// TIA Portal project "TCP Client" (V15.1)

(* hardware
DEVICE "ET 200SP station_1"  ET 200SP-Station
   slot 0: "Rack_0"  Rack  6ES5 710-8MAx1
   slot 1: "PLC_1"  CPU 1510SP F-1 PN  6ES7 510-1SJ00-0AB0  V1.8
   slot 127: "BA 2xRJ45"  BA 2xRJ45  6ES7 193-6AR00-0AA0  V0.0
      slot 32769: "Port_1"  6ES7 193-6AR00-0AA0
      slot 32770: "Port_2"  6ES7 193-6AR00-0AA0
*)

// ===== PLC "PLC_1"  CPU 1510SP F-1 PN =====

FUNCTION_BLOCK "01CommTCP"   // FB4, SCL
{ S7_Optimized_Access := 'FALSE' }
VERSION : 0.1
   VAR_INPUT
      IP1 : Byte;
      IP2 : Byte;
      IP3 : Byte;
      IP4 : Byte;
      Port : UInt;
      ConID : Conn_Ouc;
   END_VAR
   VAR
      RcvBusy : Bool;
      SndBuf : Array[1..40] of Char;
      RcvBuf : Array[1..40] of Char;
      Size : Struct
         Snd : Int;
         Rcv : Int;
      END_STRUCT;
      Connect : TCON;
      Snd : TSEND;
      Rcv : TRCV;
      SndCount : Int;
      RcvCount : Int;
      Req : Bool;
      RcvLen : Int;
      "Step" : Int;
      Zero : Int;
      RetVal : Int;
      Tout : TON_TIME;
      TON_Repeat : TON_TIME;
      DisConnect : TDISCON;
      conData : TCON_IP_v4;
      tonDelay : TON_TIME;
      tonConTout : TON_TIME;
      tonConWarning : TON_TIME;
      WarnConnection : Program_Alarm;
      wStatus : Word;
      byTestState : Byte;
      xError : Bool;
      CntOfSendBuf : UInt;
      CntOfRecBuf : UInt;
      bufferTimer : TON_TIME;
      status : Word;
      error : Bool;
   END_VAR
   VAR_TEMP
      xSig : Bool;
   END_VAR
BEGIN
   //********************************************************************************
   // Initialization
   //********************************************************************************

   CASE #Step OF

   0:
       //*********************************
       //  Init part 1 step moved to 0
       //*********************************
       #conData.InterfaceId := 64;
       #conData.ID := #ConID;
       #conData.ConnectionType := 11;
       #conData.ActiveEstablished := True;
       #conData.RemotePort := #Port;
       #conData.LocalPort := 0;
       #conData.RemoteAddress.ADDR[1] := #IP1;
       #conData.RemoteAddress.ADDR[2] := #IP2;
       #conData.RemoteAddress.ADDR[3] := #IP3;
       #conData.RemoteAddress.ADDR[4] := #IP4;
       #Step := 1;

   1:  //*********************************
       //  Init Part 2
       //*********************************
       #RcvCount := 0;
       #SndCount := 0;
       #Rcv.EN_R := False;
       #Snd.REQ := False;
       #Zero := 0;
       #RetVal := 0;

       #Connect(REQ := False, ID := #conData.ID, CONNECT := #conData);

       #DisConnect(REQ := False, ID := #conData.ID);
       #Step := 2;

   2:  // wait connection closed    
       #DisConnect(REQ := True, ID := #conData.ID);
       IF #DisConnect.DONE OR NOT #DisConnect.BUSY THEN
           #DisConnect(REQ := False, ID := #conData.ID);
           #tonDelay(IN := False, PT := t#1s);
           #Step := 3;
       END_IF;

   3:  // wait delay time
       #tonDelay(IN := True,PT := t#2s);
       IF #tonDelay.Q THEN
           #tonConTout(IN := False,PT := t#3s);
           #Step := 4;
       END_IF;


   4:  // establish connection    
       #tonConTout(IN := True, PT := t#3s);
       IF #tonConTout.Q THEN
           #Step := 1;
       END_IF;
       #Connect(REQ := True, ID := #conData.ID, CONNECT := #conData);
       IF #Connect.DONE THEN
           #Connect(REQ := False, ID := #conData.ID, CONNECT := #conData);
           #Rcv.EN_R := True;
           #Step := 5;
       END_IF;
   END_CASE;



   //------------------------------------------------------------------------------------------
   // call TCP/IP send function   
   //------------------------------------------------------------------------------------------

   #Connect(ID := #conData.ID,
            CONNECT := #conData);
   IF #Connect.DONE AND NOT #Connect.ERROR THEN
       #Connect.REQ := False;
       #Rcv.EN_R := True;
   END_IF;

   #TON_Repeat(IN := #Rcv.EN_R AND NOT #Snd.REQ,
               PT := t#100ms);
   IF #TON_Repeat.Q THEN
       #Snd.REQ := True;
   END_IF;
   // 
   // IF #Rcv.EN_R AND NOT #Snd.REQ AND "CarriageReleased" THEN
   //     #Snd.REQ := true;
   // END_IF;


   // LEN must be the length of the data you want to send

   Strg_TO_Chars(Strg := "Stringy".GlobString,
                 pChars := 0,
                 Cnt => #CntOfSendBuf,
                 Chars := #SndBuf);

   Strg_TO_Chars(Strg := "Stringy".GlobString,
                 pChars := 0,
                 Cnt => #CntOfSendBuf,
                 Chars := "Stringy".SendBuffer);

   #Snd(ID := #conData.ID,
        LEN := "SizeOf"(Ptr := #SndBuf),
        DATA := #SndBuf);

   #Rcv(ID := #conData.ID,
        LEN := 1,
        DATA := "Stringy".RecBuffer, STATUS => #status, ERROR => #error);

   Chars_TO_Strg(Chars:="Stringy".RecBuffer,
                 pChars:=0,
                 Cnt:=#CntOfRecBuf,
                 Strg=>"Stringy".GlobRecBuff);


   IF #Snd.DONE THEN
       #Snd.REQ := False;
       IF NOT #Snd.ERROR THEN
           #SndCount := #SndCount + 1;
       END_IF;
   END_IF;


   IF #Tout.Q OR #Rcv.ERROR OR #Snd.ERROR THEN
   #Step := 0;
   END_IF;
END_FUNCTION_BLOCK

ORGANIZATION_BLOCK "Main"   // OB1, LAD, ProgramCycle
TITLE = "Main Program Sweep (Cycle)"
{ S7_Optimized_Access := 'TRUE' }
VERSION : 0.1
   VAR_INPUT
      Initial_Call : Bool;   // Initial call of this OB
      Remanence : Bool;   // =True, if remanent data are available
   END_VAR
BEGIN
END_ORGANIZATION_BLOCK